FUNCTION_BLOCK PUBLIC Moving
VAR_INPUT
	Position : int;
END_VAR
VAR_OUTPUT
END_VAR
VAR
	Busy: BOOL;
	PulseTimer2: TP;
	
	BusyFtrigX : F_Trig;
	BusyFtrigY : F_Trig;
	
	ReadyX : BOOL;
	ReadyY : BOOL;
END_VAR

PulseTimer2(IN:=Busy, PT:=T#150MS);

Busy := TRUE;

CASE Position OF
	0:
		GVL_IO.INX0_from_Input0_tableX := FALSE;
		GVL_IO.INX1_from_Input1_tableX := FALSE;
		GVL_IO.INX2_from_Input2_tableX := TRUE;
		GVL_IO.INY0_from_Input0_translY := TRUE;
		GVL_IO.INY1_from_Input1_translY := FALSE;
		GVL_IO.INY2_from_Input2_translY := TRUE;
	1:
		GVL_IO.INX0_from_Input0_tableX := FALSE;
		GVL_IO.INX1_from_Input1_tableX := FALSE;
		GVL_IO.INX2_from_Input2_tableX := FALSE;
		GVL_IO.INY0_from_Input0_translY := FALSE;
		GVL_IO.INY1_from_Input1_translY := FALSE;
		GVL_IO.INY2_from_Input2_translY := FALSE;
	2:
		GVL_IO.INX0_from_Input0_tableX := TRUE;
		GVL_IO.INX1_from_Input1_tableX := FALSE;
		GVL_IO.INX2_from_Input2_tableX := FALSE;
		GVL_IO.INY0_from_Input0_translY := FALSE;
		GVL_IO.INY1_from_Input1_translY := FALSE;
		GVL_IO.INY2_from_Input2_translY := FALSE;
	3:
		GVL_IO.INX0_from_Input0_tableX := FALSE;
		GVL_IO.INX1_from_Input1_tableX := TRUE;
		GVL_IO.INX2_from_Input2_tableX := FALSE;
		GVL_IO.INY0_from_Input0_translY := FALSE;
		GVL_IO.INY1_from_Input1_translY := FALSE;
		GVL_IO.INY2_from_Input2_translY := FALSE;
	4:
		GVL_IO.INX0_from_Input0_tableX := TRUE;
		GVL_IO.INX1_from_Input1_tableX := TRUE;
		GVL_IO.INX2_from_Input2_tableX := FALSE;
		GVL_IO.INY0_from_Input0_translY := FALSE;
		GVL_IO.INY1_from_Input1_translY := FALSE;
		GVL_IO.INY2_from_Input2_translY := FALSE;
	5:
		GVL_IO.INX0_from_Input0_tableX := FALSE;
		GVL_IO.INX1_from_Input1_tableX := FALSE;
		GVL_IO.INX2_from_Input2_tableX := TRUE;
		GVL_IO.INY0_from_Input0_translY := FALSE;
		GVL_IO.INY1_from_Input1_translY := FALSE;
		GVL_IO.INY2_from_Input2_translY := FALSE;
	6:
		GVL_IO.INX0_from_Input0_tableX := FALSE;
		GVL_IO.INX1_from_Input1_tableX := FALSE;
		GVL_IO.INX2_from_Input2_tableX := FALSE;
		GVL_IO.INY0_from_Input0_translY := TRUE;
		GVL_IO.INY1_from_Input1_translY := FALSE;
		GVL_IO.INY2_from_Input2_translY := FALSE;
	7:
		GVL_IO.INX0_from_Input0_tableX := TRUE;
		GVL_IO.INX1_from_Input1_tableX := FALSE;
		GVL_IO.INX2_from_Input2_tableX := FALSE;
		GVL_IO.INY0_from_Input0_translY := TRUE;
		GVL_IO.INY1_from_Input1_translY := FALSE;
		GVL_IO.INY2_from_Input2_translY := FALSE;
	8:
		GVL_IO.INX0_from_Input0_tableX := FALSE;
		GVL_IO.INX1_from_Input1_tableX := TRUE;
		GVL_IO.INX2_from_Input2_tableX := FALSE;
		GVL_IO.INY0_from_Input0_translY := TRUE;
		GVL_IO.INY1_from_Input1_translY := FALSE;
		GVL_IO.INY2_from_Input2_translY := FALSE;
	9:
		GVL_IO.INX0_from_Input0_tableX := TRUE;
		GVL_IO.INX1_from_Input1_tableX := TRUE;
		GVL_IO.INX2_from_Input2_tableX := FALSE;
		GVL_IO.INY0_from_Input0_translY := TRUE;
		GVL_IO.INY1_from_Input1_translY := FALSE;
		GVL_IO.INY2_from_Input2_translY := FALSE;
	10:
		GVL_IO.INX0_from_Input0_tableX := FALSE;
		GVL_IO.INX1_from_Input1_tableX := FALSE;
		GVL_IO.INX2_from_Input2_tableX := TRUE;
		GVL_IO.INY0_from_Input0_translY := TRUE;
		GVL_IO.INY1_from_Input1_translY := FALSE;
		GVL_IO.INY2_from_Input2_translY := FALSE;
	11:
		GVL_IO.INX0_from_Input0_tableX := FALSE;
		GVL_IO.INX1_from_Input1_tableX := FALSE;
		GVL_IO.INX2_from_Input2_tableX := FALSE;
		GVL_IO.INY0_from_Input0_translY := FALSE;
		GVL_IO.INY1_from_Input1_translY := TRUE;
		GVL_IO.INY2_from_Input2_translY := FALSE;
	12:
		GVL_IO.INX0_from_Input0_tableX := TRUE;
		GVL_IO.INX1_from_Input1_tableX := FALSE;
		GVL_IO.INX2_from_Input2_tableX := FALSE;
		GVL_IO.INY0_from_Input0_translY := FALSE;
		GVL_IO.INY1_from_Input1_translY := TRUE;
		GVL_IO.INY2_from_Input2_translY := FALSE;
	13:
		GVL_IO.INX0_from_Input0_tableX := FALSE;
		GVL_IO.INX1_from_Input1_tableX := TRUE;
		GVL_IO.INX2_from_Input2_tableX := FALSE;
		GVL_IO.INY0_from_Input0_translY := FALSE;
		GVL_IO.INY1_from_Input1_translY := TRUE;
		GVL_IO.INY2_from_Input2_translY := FALSE;
	14:
		GVL_IO.INX0_from_Input0_tableX := TRUE;
		GVL_IO.INX1_from_Input1_tableX := TRUE;
		GVL_IO.INX2_from_Input2_tableX := FALSE;
		GVL_IO.INY0_from_Input0_translY := FALSE;
		GVL_IO.INY1_from_Input1_translY := TRUE;
		GVL_IO.INY2_from_Input2_translY := FALSE;
	15:
		GVL_IO.INX0_from_Input0_tableX := FALSE;
		GVL_IO.INX1_from_Input1_tableX := FALSE;
		GVL_IO.INX2_from_Input2_tableX := TRUE;
		GVL_IO.INY0_from_Input0_translY := FALSE;
		GVL_IO.INY1_from_Input1_translY := TRUE;
		GVL_IO.INY2_from_Input2_translY := FALSE;
	16:
		GVL_IO.INX0_from_Input0_tableX := FALSE;
		GVL_IO.INX1_from_Input1_tableX := FALSE;
		GVL_IO.INX2_from_Input2_tableX := FALSE;
		GVL_IO.INY0_from_Input0_translY := TRUE;
		GVL_IO.INY1_from_Input1_translY := TRUE;
		GVL_IO.INY2_from_Input2_translY := FALSE;
	17:
		GVL_IO.INX0_from_Input0_tableX := TRUE;
		GVL_IO.INX1_from_Input1_tableX := FALSE;
		GVL_IO.INX2_from_Input2_tableX := FALSE;
		GVL_IO.INY0_from_Input0_translY := TRUE;
		GVL_IO.INY1_from_Input1_translY := TRUE;
		GVL_IO.INY2_from_Input2_translY := FALSE;
	18:
		GVL_IO.INX0_from_Input0_tableX := FALSE;
		GVL_IO.INX1_from_Input1_tableX := TRUE;
		GVL_IO.INX2_from_Input2_tableX := FALSE;
		GVL_IO.INY0_from_Input0_translY := TRUE;
		GVL_IO.INY1_from_Input1_translY := TRUE;
		GVL_IO.INY2_from_Input2_translY := FALSE;
	19:
		GVL_IO.INX0_from_Input0_tableX := TRUE;
		GVL_IO.INX1_from_Input1_tableX := TRUE;
		GVL_IO.INX2_from_Input2_tableX := FALSE;
		GVL_IO.INY0_from_Input0_translY := TRUE;
		GVL_IO.INY1_from_Input1_translY := TRUE;
		GVL_IO.INY2_from_Input2_translY := FALSE;
	20:
		GVL_IO.INX0_from_Input0_tableX := FALSE;
		GVL_IO.INX1_from_Input1_tableX := FALSE;
		GVL_IO.INX2_from_Input2_tableX := TRUE;
		GVL_IO.INY0_from_Input0_translY := TRUE;
		GVL_IO.INY1_from_Input1_translY := TRUE;
		GVL_IO.INY2_from_Input2_translY := FALSE;
	21:
		GVL_IO.INX0_from_Input0_tableX := FALSE;
		GVL_IO.INX1_from_Input1_tableX := FALSE;
		GVL_IO.INX2_from_Input2_tableX := FALSE;
		GVL_IO.INY0_from_Input0_translY := FALSE;
		GVL_IO.INY1_from_Input1_translY := FALSE;
		GVL_IO.INY2_from_Input2_translY := TRUE;
	22:
		GVL_IO.INX0_from_Input0_tableX := TRUE;
		GVL_IO.INX1_from_Input1_tableX := FALSE;
		GVL_IO.INX2_from_Input2_tableX := FALSE;
		GVL_IO.INY0_from_Input0_translY := FALSE;
		GVL_IO.INY1_from_Input1_translY := FALSE;
		GVL_IO.INY2_from_Input2_translY := TRUE;
	23:
		GVL_IO.INX0_from_Input0_tableX := FALSE;
		GVL_IO.INX1_from_Input1_tableX := TRUE;
		GVL_IO.INX2_from_Input2_tableX := FALSE;
		GVL_IO.INY0_from_Input0_translY := FALSE;
		GVL_IO.INY1_from_Input1_translY := FALSE;
		GVL_IO.INY2_from_Input2_translY := TRUE;
	24:
		GVL_IO.INX0_from_Input0_tableX := TRUE;
		GVL_IO.INX1_from_Input1_tableX := TRUE;
		GVL_IO.INX2_from_Input2_tableX := FALSE;
		GVL_IO.INY0_from_Input0_translY := FALSE;
		GVL_IO.INY1_from_Input1_translY := FALSE;
		GVL_IO.INY2_from_Input2_translY := TRUE;
	25:
		GVL_IO.INX0_from_Input0_tableX := FALSE;
		GVL_IO.INX1_from_Input1_tableX := FALSE;
		GVL_IO.INX2_from_Input2_tableX := TRUE;
		GVL_IO.INY0_from_Input0_translY := FALSE;
		GVL_IO.INY1_from_Input1_translY := FALSE;
		GVL_IO.INY2_from_Input2_translY := TRUE;
END_CASE

		GVL_IO.DRIVEX_MOVE_tableX := PulseTimer2.Q;
		GVL_IO.DRIVEY_MOVE_translY := PulseTimer2.Q;
		
		//// Koppelen van outputs Busy aan var's. Triggered op een falling edge.
	   	BusyFtrigX ( clk := gvl_io.BUSYX_BUSY_tableX ); 
	  	BusyFtrigY ( clk := gvl_io.BUSYY_BUSY_traslationY );
		
		// Bools setten aan de hand van triggers.
		IF BusyFtrigX.Q THEN
			ReadyX:= TRUE;
		END_IF
		
		IF BusyFtrigY.Q THEN
			ReadyY:= TRUE;
		END_IF
		
		// Init voltooid ga naar idle
		IF ReadyY AND ReadyX THEN
			GVL_IO.DRIVEX_MOVE_tableX := FALSE;
			GVL_IO.DRIVEY_MOVE_translY := FALSE;
			ReadyX:= FALSE;
			ReadyY:= FALSE;
			Busy:= FALSE;
			//CurrentState := States.PickUpDown;
		END_IF

END_FUNCTION_BLOCK

(* stored: Version 1.1.0.1, ProductVersion 3.1.4022.12
   POU Moving: Id {398a761a-5c1a-4f67-95e6-29bf851a4f5a}, SpecialFunc None *)
